TYPE LG_ControlRegs :
STRUCT
	ui_OperatingMode	:	UINT := 3;
	ui_ControlMode		:	UINT := 1;
	r_Setpoint1			:	REAL := 20;
	r_RoomSetpoint		:	REAL;
	ui_TempShiftValue	:	UINT;
	r_setpoint2			:	REAL;
	r_RoomSetpoint2		:	REAL;
	ui_TempShiftValue2	:	UINT;
	r_DHWgoalTemp		:	REAL;
	ui_EnergyStatus		:	UINT := 2;	
END_STRUCT
END_TYPE

(* stored: Version 1.1.0.1, ProductVersion 3.1.4026.18
   DUT LG_ControlRegs: Id {1f0fd639-1746-464c-bfb9-b58355089f9a} *)
